// TIA Portal V19 export
VAR_GLOBAL   // PLC tag table "VLV"
END_VAR
